Staubli VAL3: SWAP.pjx

Parameters version=s7.0 stackSize=5000 millimeterUnit=true
Program file=start.pgx
Program file=stop.pgx
Data file=Swap.dtx
